FUNCTION_BLOCK FB_RecipeBuilderBorgoWings EXTENDS FB_RecipeBase

METHOD Build : BOOL
VAR_INST
    TotalY          : REAL;
    TotalX          : REAL;
    ShorterY        : REAL;
    ShorterX        : REAL;
END_VAR
TotalY   := _Config.PanelFrontLength + 2 * _Config.PanelHeight;
TotalX   := _Config.PanelFrontWidth  + 2 * _Config.PanelHeight; 
ShorterY := TotalY - _Config.PanelHeight;
ShorterX := TotalX - _Config.PanelHeight;
THIS^.UpdateNestingLimits();

IF _Config.FillAll THEN
    _ActualCopiesX := _MaxCopiesX;
    _ActualCopiesY := _MaxCopiesY;
ELSE
    // Jeśli nie "wypełnij", to bierzemy to co chce operator, ale obcinamy od 1 do Max!
    _ActualCopiesX := LIMIT(1, _Config.RequestedCopiesX, _MaxCopiesX);
    _ActualCopiesY := LIMIT(1, _Config.RequestedCopiesY, _MaxCopiesY);
END_IF


// ------------------------------------
// 1. Segregracja frezowania (Grooving)
// ------------------------------------
_SegmentsToGroove := 4;

_SegmentsGroove[1].Start.X := TotalX;
_SegmentsGroove[1].Stop.X  := 0;
_SegmentsGroove[1].Start.Y := ShorterY;
_SegmentsGroove[1].Stop.Y  := ShorterY;

_SegmentsGroove[2].Start.X := TotalX;
_SegmentsGroove[2].Stop.X  := 0; 
_SegmentsGroove[2].Start.Y := _Config.PanelHeight;
_SegmentsGroove[2].Stop.Y  := _Config.PanelHeight;

_SegmentsGroove[3].Start.X := ShorterX;
_SegmentsGroove[3].Stop.X  := ShorterX;
_SegmentsGroove[3].Start.Y := TotalY;
_SegmentsGroove[3].Stop.Y  := 0;

_SegmentsGroove[4].Start.Y := TotalY;
_SegmentsGroove[4].Stop.Y  := 0;
_SegmentsGroove[4].Start.X := _Config.PanelHeight;
_SegmentsGroove[4].Stop.X  := _Config.PanelHeight;

// ------------------------------------
// 2. Cięcie w osi X (Cut X)
// ------------------------------------
_SegmentsToCutX := 6;

// Short Box Segments
_SegmentsCutX[1].Start.X := TotalX + _Config.CuttingOverpass;
_SegmentsCutX[1].Stop.X  := ShorterX;
_SegmentsCutX[1].Start.Y := ShorterY;
_SegmentsCutX[1].Stop.Y  := ShorterY;

_SegmentsCutX[2].Start.X := _Config.PanelHeight;
_SegmentsCutX[2].Stop.X  := -_Config.CuttingOverpass;
_SegmentsCutX[2].Start.Y := ShorterY;
_SegmentsCutX[2].Stop.Y  := ShorterY;

_SegmentsCutX[3].Start.X := TotalX + _Config.CuttingOverpass;
_SegmentsCutX[3].Stop.X  := ShorterX;
_SegmentsCutX[3].Start.Y := _Config.PanelHeight;
_SegmentsCutX[3].Stop.Y  := _Config.PanelHeight;

_SegmentsCutX[4].Start.X := _Config.PanelHeight;
_SegmentsCutX[4].Stop.X  := -_Config.CuttingOverpass;
_SegmentsCutX[4].Start.Y := _Config.PanelHeight;
_SegmentsCutX[4].Stop.Y  := _Config.PanelHeight;

// Panel Dimensions Shorter Flaps
_SegmentsCutX[5].Start.X := TotalX + _Config.CuttingOverpass;
_SegmentsCutX[5].Stop.X  := -_Config.CuttingOverpass;
_SegmentsCutX[5].Start.Y := TotalY - _Config.RailHeightCorrection;
_SegmentsCutX[5].Stop.Y  := TotalY - _Config.RailHeightCorrection;

_SegmentsCutX[6].Start.X := TotalX + _Config.CuttingOverpass;
_SegmentsCutX[6].Stop.X  := -_Config.CuttingOverpass;
_SegmentsCutX[6].Start.Y := _Config.RailHeightCorrection;
_SegmentsCutX[6].Stop.Y  := _Config.RailHeightCorrection;

// ------------------------------------
// 3. Cięcie w osi Y (Cut Y)
// ------------------------------------
_SegmentsToCutY := 6;

// Short Box Segments
_SegmentsCutY[1].Start.X := ShorterX;
_SegmentsCutY[1].Stop.X  := ShorterX;
_SegmentsCutY[1].Start.Y := TotalY + _Config.CuttingOverpass;
_SegmentsCutY[1].Stop.Y  := ShorterY;

_SegmentsCutY[2].Start.X := _Config.PanelHeight;
_SegmentsCutY[2].Stop.X  := _Config.PanelHeight;
_SegmentsCutY[2].Start.Y := TotalY + _Config.CuttingOverpass;
_SegmentsCutY[2].Stop.Y  := ShorterY;

_SegmentsCutY[3].Start.X := ShorterX;
_SegmentsCutY[3].Stop.X  := ShorterX;
_SegmentsCutY[3].Start.Y := _Config.PanelHeight;
_SegmentsCutY[3].Stop.Y  := -_Config.CuttingOverpass;

_SegmentsCutY[4].Start.X := _Config.PanelHeight;
_SegmentsCutY[4].Stop.X  := _Config.PanelHeight;
_SegmentsCutY[4].Start.Y := _Config.PanelHeight;
_SegmentsCutY[4].Stop.Y  := -_Config.CuttingOverpass;

// Panel Dimensions
_SegmentsCutY[5].Start.X := TotalX;
_SegmentsCutY[5].Stop.X  := TotalX;
_SegmentsCutY[5].Start.Y := TotalY + _Config.CuttingOverpass;
_SegmentsCutY[5].Stop.Y  := -_Config.CuttingOverpass;

_SegmentsCutY[6].Start.X := 0;
_SegmentsCutY[6].Stop.X  := 0;
_SegmentsCutY[6].Start.Y := TotalY + _Config.CuttingOverpass;
_SegmentsCutY[6].Stop.Y  := -_Config.CuttingOverpass;


Build := TRUE;
END_METHOD

METHOD FB_init : BOOL
VAR_INPUT
	bInitRetains : BOOL; // if TRUE, the retain variables are initialized (warm start / cold start)
	bInCopyCode : BOOL;  // if TRUE, the instance afterwards gets moved into the copy code (online change)
END_VAR
_Limits.PanelFrontLength.MinVal := 100.0;
_Limits.PanelFrontLength.MaxVal := 1234.0;

_Limits.PanelFrontWidth.MinVal  := 100.0;
_Limits.PanelFrontWidth.MaxVal  := 1234.0;

_Limits.PanelHeight.MinVal      := 0.0;
_Limits.PanelHeight.MaxVal      := 1234.0;

_Limits.RailHeightCorrection.MinVal := 12.0;
_Limits.RailHeightCorrection.MaxVal := 14.0;

_Limits.CuttingOverpass.MinVal := 0.0;
_Limits.CuttingOverpass.MaxVal := 50.0;

_Limits.GroovingOverpass.MinVal := 0.0;
_Limits.GroovingOverpass.MaxVal := 50.0;
END_METHOD

END_FUNCTION_BLOCK

(* stored: Version 1.1.0.1, ProductVersion 3.1.4024.15
   POU FB_RecipeBuilderBorgoWings: Id {3f83a514-1f2f-4e3d-921c-ca7c0b60e17f}, SpecialFunc None
   Method Build: Id {c08ade7c-db75-4c50-8457-5bb392619adf}
   Method FB_init: Id {166bcf26-5e69-4b30-9881-84478d8b0138} *)
